KUKA KRL data list: Up113.dat

&ACCESS RVP1
&COMMENT Wartung Greifer 2 VW310-6
&PARAM DISKPATH = KRC:\R1\UPs
&PARAM TEMPLATE = C:\KRC\Roboter\Template\upvorgabe
&PARAM EDITMASK = Up999[1-999]
&PARAM TPVW_VERSION = 8.1.8
DEFDAT UP113
; FOLD ;%{H} %MKUKATPVW
; ENDFOLD
; interface to basic routines
 EXT  BAS (BAS_COMMAND  :IN,REAL  :IN )
; interface to VW-standard routines
EXT VW (VW_COMMAND:IN, BOOL: IN, REAL:IN, REAL:IN, REAL:IN, REAL:IN, BOOL :IN, E6POS :IN )
; interface to VW_USER - Call
EXT  VW_USER (VW_USER_CMD :IN,INT :IN,REAL  :IN,REAL  :IN,REAL  :IN,REAL  :IN,REAL  :IN,REAL  :IN,BOOL  :IN )
EXT  VW_USR_R (VW_USER_CMD :IN,INT :IN,REAL  :IN,REAL  :IN,REAL  :IN,REAL  :IN,REAL  :IN,REAL  :IN,BOOL  :IN )
EXT  IBGN (IBGN_COMMAND  :IN,BOOL  :IN,REAL  :IN,REAL  :IN,BOOL  :IN,E6POS  :OUT )
; interface select routine
EXTFCT INT  SELECT (SUBTYPE  :IN,INT  :IN,BOOL  :IN,ARI_TYP  :IN,INT  :IN,BOOL_TYP  :IN,INT  :IN,BOOL  :IN)
INT VW_NEXT_FREE = 6
INT VW_NFREE_SPS = 6
INT VW_MAX_SPS = 106
DECL VW_MPARA_TYP P1_D = {TOOL_NO 7,BASE_NO 0,VB 100,VE 0,ACC 100,TRG_TIME 0,MOVE_TYPE #PTP_MOTION}
DECL E6POS P1 = {X 1564.05, Y -372.63, Z 2140.98, A 0.001, B 29.999, C 89.9, S 2, T 42 , E1 0.0, E2 0.0, E3 0.0, E4 0.0, E5 0.0, E6 0.0}
DECL VW_MPARA_TYP P2_D = {TOOL_NO 7,BASE_NO 0,VB 100,VE 100,ACC 100,TRG_TIME 0,MOVE_TYPE #PTP_MOTION}
DECL E6POS P2 = {X 2454.9, Y -276.25, Z 532.75, A -1.871, B 65.317, C 179.086, S 2, T 42 , E1 0.0, E2 0.0, E3 0.0, E4 0.0, E5 0.0, E6 0.0}
DECL VW_MPARA_TYP P3_D = {TOOL_NO 7,BASE_NO 0,VB 100,VE 0,ACC 100,TRG_TIME 5,MOVE_TYPE #PTP_MOTION}
DECL E6POS P3 = {X 2408.5, Y -273.32, Z -507.74, A 21.298, B 88.265, C -157.595, S 2, T 42 , E1 0.0, E2 0.0, E3 0.0, E4 0.0, E5 0.0, E6 0.0}
DECL VW_MPARA_TYP P4_D = {TOOL_NO 7,BASE_NO 0,VB 100,VE 100,ACC 100,TRG_TIME 0,MOVE_TYPE #PTP_MOTION}
DECL E6POS P4 = {X 2454.89, Y -276.25, Z 532.75, A -1.871, B 65.317, C 179.086, S 2, T 42 , E1 0.0, E2 0.0, E3 0.0, E4 0.0, E5 0.0, E6 0.0}
DECL VW_MPARA_TYP P5_D = {TOOL_NO 7,BASE_NO 0,VB 100,VE 0,ACC 100,TRG_TIME 0,MOVE_TYPE #PTP_MOTION}
DECL E6POS P5 = {X 1564.05, Y -372.63, Z 2140.98, A 0.001, B 29.999, C 89.9, S 2, T 42 , E1 0.0, E2 0.0, E3 0.0, E4 0.0, E5 0.0, E6 0.0}
ENDDAT
